TYPE E_PositionState :
(
RETRACTED    := 0,
INSERTED    := 1,
MOVING    := 2,
INVALID :=3
);
END_TYPE

(* stored: Version 1.1.0.1
   DUT E_PositionState: Id {61a5e714-50c7-4f12-a7ea-a0cbcc21a898} *)
